(* IEC 61131-3 sources: eCockpitGit/test_project/src/%F%02 System/%F%03 LoadSaveManager/%POU%FB_LoadSave, 3 files *)

(* ---- %METH%logChange.st ---- *)
//This adds the path for the log
// |**Version**|**Author**| **Date** |**Changes**
// | 1         | NSN      | 19-09-20 | Creation
METHOD PROTECTED logChange
VAR_INPUT
	valType			:ESysType;
	valPoint		:POINTER TO USysTypes;
END_VAR
VAR
	i				:BYTE;
	levelBuffer		:BYTE;
	stringBuffer	:STRING(200);
///	logBuffer		:STRING(Logs.modLogBufferSize);
	writer			:FB_JSONWriter;
	lenght			:WORD;
END_VAR
(*%!%__DELIMITER__%!%*)
IF doLogInt THEN
	IF selectedType = EStructType.tArray THEN
		keyFound	:=		reader.nextArray() <> EStructType.none;
	END_IF
	IF NOT(dontLog) AND keyFound THEN
		CASE valType OF
			ESysType.tBool:
				IF reader.valueType = EStructType.tBool AND_THEN valPoint^.bBOOL = reader.readBool() THEN
					RETURN;
				END_IF

			//Bytes
			ESysType.tBYTE,ESysType.tUSINT:
				IF reader.valueType = EStructType.number AND_THEN valPoint^.bBYTE = reader.readDword() THEN
					RETURN;
				END_IF

			ESysType.tWORD,ESysType.tUINT:
				IF reader.valueType = EStructType.number AND_THEN valPoint^.bWORD = reader.readDword() THEN
					RETURN;
				END_IF

			ESysType.tDWORD,ESysType.tUDINT:
				IF reader.valueType = EStructType.number AND_THEN valPoint^.bDWORD = reader.readDword() THEN
					RETURN;
				END_IF

			//INTs
			ESysType.tSINT:
				IF reader.valueType = EStructType.number AND_THEN valPoint^.bSINT = reader.readDint() THEN
					RETURN;
				END_IF
			ESysType.tINT:
				IF reader.valueType = EStructType.number AND_THEN valPoint^.bINT = reader.readDint() THEN
					RETURN;
				END_IF
			ESysType.tDINT:
				IF reader.valueType = EStructType.number AND_THEN valPoint^.bDINT = reader.readDint() THEN
					RETURN;
				END_IF

			ESysType.tReal:
				IF reader.valueType = EStructType.number AND_THEN valPoint^.bREAL = reader.readReal() THEN
					RETURN;
				END_IF
			ESysType.tNONE:
				IF reader.valueType = EStructType.null THEN
					RETURN;
				END_IF
			ESysType.tString:
				IF reader.valueType = EStructType.tString AND_THEN reader.compareString(str:=valPoint) THEN
					RETURN;
				END_IF
		END_CASE

///		writer.Initialize(buffer:=ADR(logBuffer),bufferSize:=Logs.modLogBufferSize,singleLine:=TRUE,bottomType:=EStructType.object);

		writer.addKey(name:=GTSmall.Stime);
		writer.writeString(value:=GMod.modMan.S_currentTime);

		writer.addKey(name:=GTSmall.Stype);
		writer.writeString(value:=GTSmall.Schanged);

		IF module <> 0 THEN
			writer.addKey(name:=GTSmall.Suid);
			writer.writeWord(value:=module^._UID);
		END_IF

		levelBuffer		:=		reader.amountLevels;
		IF levelBuffer > 0 THEN
			writer.addKey(name:=GTSmall.Spath);
			writer.arrayStart(singleLine:=TRUE);
			FOR i := 1 TO levelBuffer DO
				reader.readKeyNameLevel(name:=ADR(stringBuffer),lenMax:=SIZEOF(stringBuffer)-1,level:=i,len=>lenght);
				IF writer.bufferLeft > lenght + 250 THEN
					writer.writeString(value:=ADR(stringBuffer));
				END_IF
			END_FOR
			writer.structEnd();
		END_IF

		writer.addKey(name:=GTSmall.Sold);
		CASE reader.valueType OF
			EStructType.tBool:
				writer.writeBool(value:=reader.readBool());
			EStructType.number:
				reader.readString(str:=ADR(stringBuffer),lenMax:=SIZEOF(stringBuffer) - 1);
				writer.writeRaw(ADR(stringBuffer));
			EStructType.null:
				writer.writeNull();
			EStructType.tString:
				reader.readString(str:=ADR(stringBuffer),lenMax:=SIZEOF(stringBuffer) - 1);
				writer.writeString(value:=ADR(stringBuffer));
		END_CASE

		writer.addKey(name:=GTSmall.Snew);
		CASE valType OF
			ESysType.tBool:
				writer.writeBool(value:=valPoint^.bBOOL);
			//Bytes
			ESysType.tBYTE,ESysType.tUSINT:
				writer.writeDword(value:=valPoint^.bBYTE);
			ESysType.tWORD,ESysType.tUINT:
				writer.writeDword(value:=valPoint^.bWORD);
			ESysType.tDWORD,ESysType.tUDINT:
				writer.writeDword(value:=valPoint^.bDWORD);

			//INTs
			ESysType.tSINT:
				writer.writeDint(value:=valPoint^.bSINT);
			ESysType.tINT:
				writer.writeDint(value:=valPoint^.bINT);
			ESysType.tDINT:
				writer.writeDint(value:=valPoint^.bDINT);

			ESysType.tReal:
				writer.writeReal(value:=valPoint^.bREAL);
			ESysType.tNONE:
				writer.writeNull();
			ESysType.tString:
				writer.writeString(value:=valPoint);
		END_CASE

		writer.deinitialize();

		//writer.writeFile(path:=Logs.moduleLog.addLog());
	END_IF
END_IF

(* ---- %METH%LSEnd.st ---- *)
//This method ends the manager, by deinitialisint XML blocks and writing to file if needed
// |**Version**|**Author**| **Date** |**Changes**
// | 1         | NSN      | 26-06-18 | Creation
// | 2         | NSN      | 31-01-19 | Updated to new standard
METHOD LSEnd
VAR
	fileResultCode			:SysTypes.RTS_IEC_RESULT;
	fileHandle				:SysTypes.RTS_IEC_HANDLE;
	sizeBuffer				:DWORD;
END_VAR
(*%!%__DELIMITER__%!%*)
IF started THEN
	IF readWrite THEN
		writer.deinitialize();
		fileHandle		:=		SysFile.SysFileOpen(szFile:=filePath,am:=SysFile.ACCESS_MODE.AM_APPEND_PLUS,pResult:=ADR(fileResultCode));
		IF fileHandle <> 0 AND fileResultCode = 0 THEN
			SysFile.SysFileSetPos(hFile:=fileHandle,ulOffset:=0);
			sizeBuffer	:=		writer.bufferSize;
			SysFile.SysFileWrite(hFile:=fileHandle,pbyBuffer:=writeBuffer,ulSize:=sizeBuffer,pResult:=ADR(fileResultCode));
			SysFile.SysFileTruncate(hFile:=fileHandle,ulSizeNew:=sizeBuffer);
			SysFile.SysFileClose(hFile:=fileHandle);
		END_IF
	END_IF
	reader.deinitialize();
	filePath			:=		'';
	readWrite			:=		FALSE;
	started				:=		FALSE;
END_IF

(* ---- %METH%LSStart.st ---- *)
//This initializes the manager with the correct values
//Returns code for result, 0 = OK, 1 = File doesn't exist, but created, 2 = File doesn't exist, 3 = File doesn't exist, and cannot be created, 4 = Unknown file error
// |**Version**|**Author**| **Date** |**Changes**
// | 1         | NSN      | 05-06-18 | Creation
METHOD LSStart: SLMResult
VAR_INPUT
	sFilePath			:APath;				//Path to save file
	xReadWrite			:BOOL;				//Set False when reading data, True when writing data
	dontLog				:BOOL;
END_VAR
VAR
	amountRead			:UDINT;
	fileResultCode		:SysTypes.RTS_IEC_RESULT;
	fileHandle			:SysTypes.RTS_IEC_HANDLE;
	fileFound			:BOOL;
END_VAR
(*%!%__DELIMITER__%!%*)
IF sFilePath <> '' AND NOT(started) THEN
	fileFound					:=		FALSE;
	//Check if file already exists
	IF FU_checkFileExists(path := sFilePath) THEN
		fileFound				:=		TRUE;
	ELSE
		LSStart.success			:=		FALSE;
		LSStart.code			:=		ERCodes.FB_LoadSave_LSStart;
		LSStart.reason			:=		GTErrors.EfileDoesntExist;
	END_IF
	//When reading a found file is needed, when writing or simulating no file is needed
	IF LSStart.success OR xReadWrite THEN
		filePath				:=		sFilePath;
		readWrite				:=		xReadWrite;
		started					:=		TRUE;
		logCorrection			:=		0;
		//The file is offloaded into the readbuffer
		IF NOT(xReadWrite) OR NOT(dontLog) THEN
			fileHandle			:=		SysFile.SysFileOpen(szFile:=sFilePath,am:=SysFile.ACCESS_MODE.AM_READ,pResult:=ADR(fileResultCode));
			IF fileHandle <> 0 AND TO_DWORD(fileHandle) <> 4294967295 AND fileResultCode = 0 THEN
				SysFile.SysFileSetPos(hFile:=fileHandle,ulOffset:=0);
				amountRead		:=		SysFile.SysFileRead(hFile:=fileHandle,pbyBuffer:=readBuffer,ulSize:=readSize,pResult:=ADR(fileResultCode));
				SysFile.SysFileClose(hFile:=fileHandle);
			END_IF
			reader.Initialize(buffer:=readBuffer,bufferSize:=readSize);
			doLogInt			:=		TRUE;
		ELSE
			fileFound			:=		FALSE;
		END_IF
		//When writing files the write buffer is initialized
		IF readWrite THEN
			writer.Initialize(buffer:=writeBuffer,bufferSize:=writeSize,singleLine:=FALSE,bottomType:=EStructType.object);
		END_IF
	END_IF
END_IF
